// TIA Portal V20 export
// export: Created 2026-07-10T11:12:32.491073Z, ExportSetting WithDefaults, DisplayName Totally Integrated Automation Portal, DisplayVersion V20, DisplayName TIA Portal Openness, DisplayVersion V20, DisplayName TIA Portal Version Control Interface, DisplayVersion V20, DisplayName STEP 7 Professional, DisplayVersion V20, DisplayName STEP 7 Safety, DisplayVersion V20, DisplayName WinCC Basic/Comfort/Advanced, DisplayVersion V20, DisplayName WinCC Unified, DisplayVersion V20
FUNCTION_BLOCK "WorkModeCycle"   // FB2, SCL
{ S7_Optimized_Access := 'TRUE' }
VERSION : 0.1
// stored: AutoNumber true, IsIECCheckEnabled false, IsRetainMemResEnabled false, MemoryReserve 100, SetENOAutomatically false, UDAEnableTagReadback false
   VAR
      "step" : Int;
      tod : Time_Of_Day;
      "return" : Int;
      dtl : DTL;
      "time" : Time;
      fracDay : Real;
   END_VAR
BEGIN
   #step := 0;

   "MB".Table.LevelRCV1Min:="MB".Table.LevelRCV1BasicMin;
   "MB".Table.LevelRCV1Max:="MB".Table.LevelRCV1BasicMax;
   "MB".Table.LevelRCV2Min:="MB".Table.LevelRCV2BasicMin;
   "MB".Table.LevelRCV2Max:="MB".Table.LevelRCV2BasicMax;

   "MB".Table.CycleStatus := 0;

   "MB".Table.RestTimeC1 := 0;
   "MB".Table.RestTimeC2 := 0;
   "MB".Table.RestTimeC3 := 0;
   "MB".Table.RestTimeC4 := 0;
   "MB".Table.RestTimeC5 := 0;

   #return := RD_LOC_T(#dtl);
   #tod := DTL_TO_TOD(#dtl);
   #time := TOD_TO_TIME(#tod);

   #fracDay := DINT_TO_REAL(#time) / 86400000.0;

   IF "MB".Table.HMI_CycleOn THEN
       IF "MB".Table.CycleDay >= "MB".Table.CycleStartDay[4] THEN
           #step := 4;
           "MB".Table.CycleStatus.%X4 := 1;
       ELSIF "MB".Table.CycleDay >= "MB".Table.CycleStartDay[3] THEN
           #step := 3;
           "MB".Table.CycleStatus.%X3 := 1;
       ELSIF "MB".Table.CycleDay >= "MB".Table.CycleStartDay[2] THEN
           #step := 2;
           "MB".Table.CycleStatus.%X2 := 1;
       ELSIF "MB".Table.CycleDay>="MB".Table.CycleStartDay[1] THEN
           #step := 1;
           "MB".Table.CycleStatus.%X1 := 1;
       ELSE
           #step := 0;
           "MB".Table.CycleStatus.%X0 := 1;
       END_IF;




       "MB".Table.LevelRCV1Min := "MB".Table.LevelRCVCycle[#step].Min;
       "MB".Table.LevelRCV2Min := "MB".Table.LevelRCVCycle[#step].Min;
       "MB".Table.LevelRCV1Max := "MB".Table.LevelRCVCycle[#step].Max;
       "MB".Table.LevelRCV2Max := "MB".Table.LevelRCVCycle[#step].Max;

       IF #step <> 4 THEN
           IF "MB".Table.CycleStartDay[#step + 1] - "MB".Table.CycleDay = 1 THEN
               "MB".Table.LevelRCV1Min := #fracDay * ("MB".Table.LevelRCVCycle[#step + 1].Min - "MB".Table.LevelRCVCycle[#step].Min) + "MB".Table.LevelRCVCycle[#step].Min;
               "MB".Table.LevelRCV1Max := #fracDay * ("MB".Table.LevelRCVCycle[#step + 1].Max - "MB".Table.LevelRCVCycle[#step].Max) + "MB".Table.LevelRCVCycle[#step].Max;
               "MB".Table.LevelRCV2Min := #fracDay * ("MB".Table.LevelRCVCycle[#step + 1].Min - "MB".Table.LevelRCVCycle[#step].Min) + "MB".Table.LevelRCVCycle[#step].Min;
               "MB".Table.LevelRCV2Max := #fracDay * ("MB".Table.LevelRCVCycle[#step + 1].Max - "MB".Table.LevelRCVCycle[#step].Max) + "MB".Table.LevelRCVCycle[#step].Max;
           END_IF;
       END_IF;



       "MB".Table.RestTimeC1:= MAX(IN1 :="MB".Table.CycleStartDay[1]-"MB".Table.CycleDay, IN2 := 0);
       "MB".Table.RestTimeC2:= MAX(IN1 :="MB".Table.CycleStartDay[2]-"MB".Table.CycleDay, IN2 := 0);
       "MB".Table.RestTimeC3:= MAX(IN1 :="MB".Table.CycleStartDay[3]-"MB".Table.CycleDay, IN2 := 0);
       "MB".Table.RestTimeC4:= MAX(IN1 :="MB".Table.CycleStartDay[4]-"MB".Table.CycleDay, IN2 := 0);
       "MB".Table.RestTimeC5 := 9999;
   END_IF;
END_FUNCTION_BLOCK
